TYPE (* IEC61131-3, Table 14#5 *)
  (* Standard: 1131-3 *)
  (* Version 0.0, 1/8/2024, Cheyan, Schneider Electric, Template *)
  PACKAGE Main;
  {SET_ATTRIBUTE(nxtDataType, ZOG1cSCbfcZvft1u0Zk0T+6RcAUOKzI+HCO0qGy87ENVHb2SavOD4qrJdexiKbsNkaNLe6SP1PUpWOrB5ucndkIXf/Atxz/dVqr3qnJqGpc74K+J7i/JR3dE4a2Owyer/cgvjbDWir76nILah0A/bA==)}
  SAV_LREAL_DINT : STRUCT
    instMag : AnalogueValue;
    q : Quality;
  END_STRUCT;
END_TYPE
